PROGRAM PnPstorageMemory_Arm
VAR
	fbGnrProductRecipeMemory_Main: fbV2_GnrProductRecipeMemory;
	tProductRecipeClearPb : TON;
END_VAR

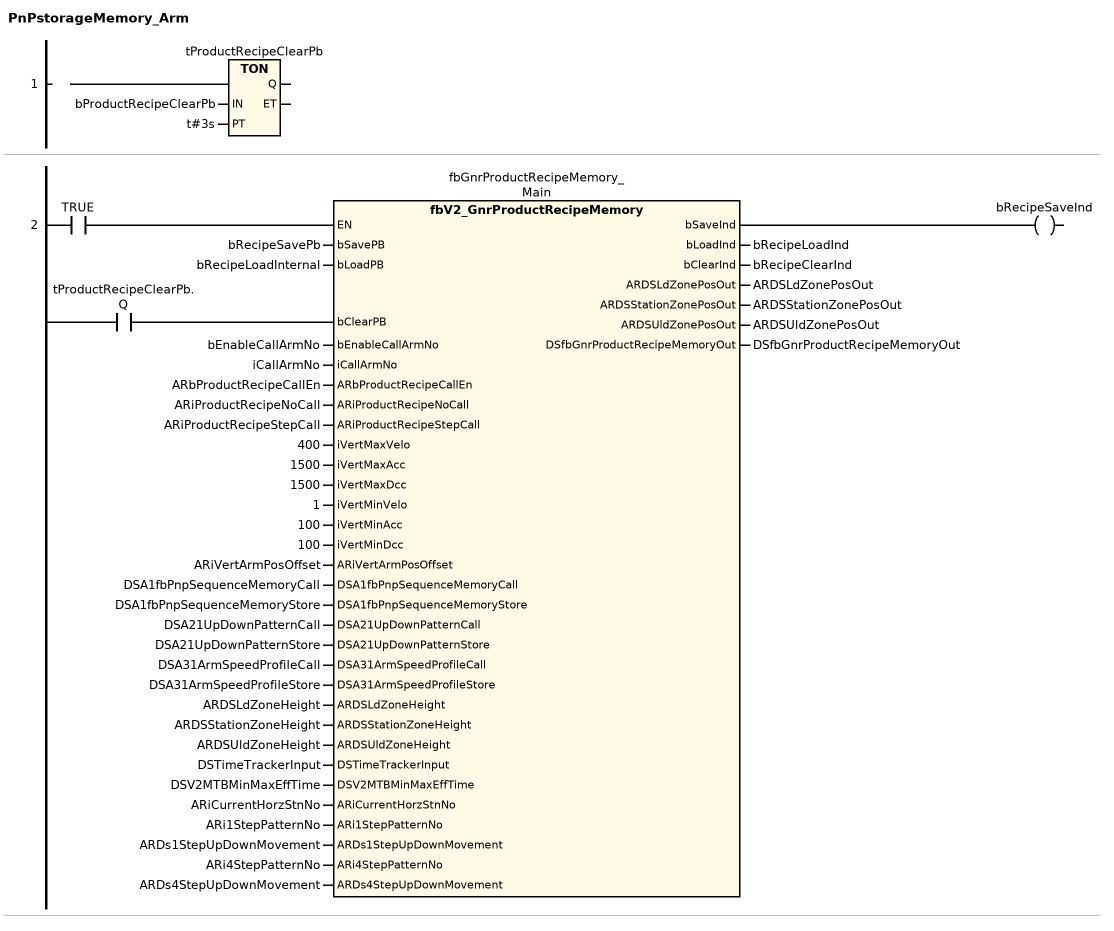
// NETWORK 1
tProductRecipeClearPb(IN := bProductRecipeClearPb, PT := t#3s); // TON

// NETWORK 2
fbGnrProductRecipeMemory_Main(
    bSavePB := bRecipeSavePb,
    bLoadPB := bRecipeLoadInternal,
    bClearPB := tProductRecipeClearPb.Q,
    bEnableCallArmNo := bEnableCallArmNo,
    iCallArmNo := iCallArmNo,
    ARbProductRecipeCallEn := ARbProductRecipeCallEn,
    ARiProductRecipeNoCall := ARiProductRecipeNoCall,
    ARiProductRecipeStepCall := ARiProductRecipeStepCall,
    iVertMaxVelo := 400,
    iVertMaxAcc := 1500,
    iVertMaxDcc := 1500,
    iVertMinVelo := 1,
    iVertMinAcc := 100,
    iVertMinDcc := 100,
    ARiVertArmPosOffset := ARiVertArmPosOffset,
    DSA1fbPnpSequenceMemoryCall := DSA1fbPnpSequenceMemoryCall,
    DSA1fbPnpSequenceMemoryStore := DSA1fbPnpSequenceMemoryStore,
    DSA21UpDownPatternCall := DSA21UpDownPatternCall,
    DSA21UpDownPatternStore := DSA21UpDownPatternStore,
    DSA31ArmSpeedProfileCall := DSA31ArmSpeedProfileCall,
    DSA31ArmSpeedProfileStore := DSA31ArmSpeedProfileStore,
    ARDSLdZoneHeight := ARDSLdZoneHeight,
    ARDSStationZoneHeight := ARDSStationZoneHeight,
    ARDSUldZoneHeight := ARDSUldZoneHeight,
    DSTimeTrackerInput := DSTimeTrackerInput,
    DSV2MTBMinMaxEffTime := DSV2MTBMinMaxEffTime,
    ARiCurrentHorzStnNo := ARiCurrentHorzStnNo,
    ARi1StepPatternNo := ARi1StepPatternNo,
    ARDs1StepUpDownMovement := ARDs1StepUpDownMovement,
    ARi4StepPatternNo := ARi4StepPatternNo,
    ARDs4StepUpDownMovement := ARDs4StepUpDownMovement,
    bLoadInd => bRecipeLoadInd,
    bClearInd => bRecipeClearInd,
    ARDSLdZonePosOut => ARDSLdZonePosOut,
    ARDSStationZonePosOut => ARDSStationZonePosOut,
    ARDSUldZonePosOut => ARDSUldZonePosOut,
    DSfbGnrProductRecipeMemoryOut => DSfbGnrProductRecipeMemoryOut); // fbV2_GnrProductRecipeMemory
bRecipeSaveInd := fbGnrProductRecipeMemory_Main.bSaveInd;

END_PROGRAM

(* stored: Version 1.1.0.1, ProductVersion 3.1.4024.12
   POU PnPstorageMemory_Arm: Id {6551c864-874a-4270-b423-7a07a3465a22}, SpecialFunc None *)
